{attribute 'no_explicit_call' := 'do not call this FB directly'}{attribute 'enable_dynamic_creation'}
FUNCTION_BLOCK FINAL IntLiteralNode EXTENDS Node
VAR
	value : _INT(0);
	out : _INT(0);
END_VAR

METHOD PUBLIC Clone : I_Node
VAR
	pNode : POINTER TO IntLiteralNode;
END_VAR
pNode := __NEW(IntLiteralNode);
Clone := pNode^;
END_METHOD

METHOD FB_init : BOOL
VAR_INPUT
	bInitRetains : BOOL; // if TRUE, the retain variables are initialized (warm start / cold start)
	bInCopyCode : BOOL;  // if TRUE, the instance afterwards gets moved into the copy code (online change)
END_VAR
AddParameter('value', value);
AddOutput('out', out);
END_METHOD

METHOD PROTECTED OnExecute : HRESULT
VAR
END_VAR
out.value := value.value;
END_METHOD

END_FUNCTION_BLOCK

(* stored: Version 1.1.0.1, ProductVersion 3.1.4024.12
   POU IntLiteralNode: Id {3c5e5a9f-b0d5-0211-16fd-53bc97fa596d}, SpecialFunc None
   Folder Constructor: Id {9b909a27-4d46-05df-3ce3-6399c4b1f252}
   Method Clone: Id {67a9183c-07aa-0faa-2114-ed0818031f17}
   Method FB_init: Id {83a363c4-3f00-0a22-306f-a55449e448d6}
   Method OnExecute: Id {59e9e693-2ba9-0063-0efe-fe1e3fa22ec2} *)
